INTERFACE ITF_ControlElement

END_INTERFACE

(* stored: Version 1.1.0.1, ProductVersion 3.1.4024.15
   Itf ITF_ControlElement: Id {877b1e1f-83e8-44f6-8ffa-51e9467885b8} *)
